{attribute 'TcGenerated'}
{attribute 'no-analysis'}
{attribute 'linkalways'}
// This function has been automatically generated from the project information.
VAR_GLOBAL CONSTANT
	{attribute 'const_non_replaced'}
	stLibVersion_TcCylinder : ST_LibVersion := (iMajor := 2, iMinor := 1, iBuild := 0, iRevision := 0, nFlags := 0, sVersion := '2.1.0');
END_VAR

(* stored: Version 1.1.0.1, ProductVersion 3.1.4026.17
   GVL Global_Version: Id {5d0cbe78-f54f-4b6f-938e-5e0c855fa3e0} *)
